TYPE ST_FlowMeterInputScaling :
STRUCT
	fMaxInputValue : LREAL;
	fMinInputValue : LREAL;
	fNeutralInputValue : LREAL;
	fNeutralDeadband : LREAL;
	fMaxOutputValue : LREAL;
	fMinOutputValue : LREAL;
	fNeutralOutputValue : LREAL;
END_STRUCT
END_TYPE

(* stored: Version 1.1.0.1, ProductVersion 3.1.4024.12
   DUT ST_FlowMeterInputScaling: Id {683501c9-0d8d-4bed-9f22-9711d203069f} *)
